// TIA Portal V17 export
// export: Created 2025-03-05T08:02:20.4169739Z, ExportSetting WithDefaults, DisplayName Totally Integrated Automation Portal, DisplayVersion V17 Update 8, DisplayName TIA Portal Openness, DisplayVersion V17 Update 8, DisplayName TIA Portal Version Control Interface, DisplayVersion V17, DisplayName SINAMICS Startdrive Advanced, DisplayVersion V17 SP2, DisplayName SINAMICS Startdrive G110M, G120, G120C, G120D, G120P, G115D, DisplayVersion V17 SP2, DisplayName SINAMICS Startdrive G130, G150, S120, S150, SINAMICS MV, S210, DisplayVersion V17 SP2, DisplayName STEP 7 Professional, DisplayVersion V17 Update 8, DisplayName SINUMERIK ONE STEP 7 Toolbox, DisplayVersion V17 Update 12, DisplayName SINUMERIK 840D sl STEP 7 Toolbox, DisplayVersion V17 Update 12, DisplayName STEP 7 Safety, DisplayVersion V17 Update 6, DisplayName WinCC Advanced, DisplayVersion V17 Update 8
TYPE "OPEN_CLOSE"
// stored: IsFailsafeCompliant false
   STRUCT
      CLOSED_PART_A_I : Bool;   // ADVANCED PART "A" INPUT / CLOSED PART A INPUT
      CLOSED_PART_B_I : Bool;   // ADVANCED PART "B" INPUT / CLOSED PART B INPUT
      CLOSED_PART_C_I : Bool;   // ADVANCED PART "C" INPUT / CLOSED PART C INPUT
      CLOSED_PART_D_I : Bool;   // ADVANCED PART "D" INPUT / CLOSED PART D INPUT
      CLOSED_PRESSURE_SW_1_I : Bool;   // ADVANCED PRESSURE SWITCH 1 / CLOSED PRESSURE SWITCH 1 INPUT
      CLOSED_PRESSURE_SW_2_I : Bool;   // ADVANCED PRESSURE SWITCH 2 / CLOSED PRESSURE SWITCH 2 INPUT
      OPEN_PART_A_I : Bool;   // RETURNED PART "A" INPUT / OPEN PART A INPUT
      OPEN_PART_B_I : Bool;   // RETURNED PART "B" INPUT / OPEN PART B INPUT
      OPEN_PART_C_I : Bool;   // RETURNED PART "C" INPUT / OPEN PART C INPUT
      OPEN_PART_D_I : Bool;   // RETURNED PART "D" INPUT / OPEN PART D INPUT
      OPEN_PRESSURE_SW_1_I : Bool;   // RETURNED PRESSURE SWITCH 1 / OPEN PRESSURE SWITCH 1 INPUT
      OPEN_PRESSURE_SW_2_I : Bool;   // RETURNED PRESSURE SWITCH 2 / OPEN PRESSURE SWITCH 2 INPUT
      CLOSED_LOW_PRESSURE_SW_I : Bool;   // CLOSED LOW PRESSURE SWITCH INPUT
      OPEN_LOW_PRESSURE_SW_I : Bool;   // OPEN LOW PRESSURE SWITCH INPUT
      ANY_CLOSED : Bool;   // ANY CLOSED INPUT
      ANY_OPEN : Bool;   // ANY OPEN INPUT
      GENERAL_CONDITIONS : Bool;   // GENERAL CONDITIONS
      CLOSE_CONDITIONS : Bool;   // ADVANCE CONDITIONS / CLOSE CONDITIONS
      OPEN_CONDITIONS : Bool;   // RETURN CONDITIONS / OPEN CONDITIONS
      RELEASE_PRESSURE_CONDITIONS : Bool;   // RELIEVE PRESSURE CONDITIONS / RELEASE PRESSURE CONDITIONS
      LOW_PRESSURE_CONDITIONS : Bool;   // RELIEVE PRESSURE CONDITIONS / LOW PRESSURE CONDITIONS
      GENERAL_CONDITIONS_HELP : Bool;   // GENERAL CONDITIONS HELP
      CLOSE_CONDITIONS_HELP : Bool;   // CLOSE CONDITIONS HELP
      OPEN_CONDITIONS_HELP : Bool;   // OPEN CONDITIONS HELP
      RELEASE_PRESSURE_CONDITIONS_HELP : Bool;   // RELEASE PRESSURE CONDITIONS HELP
      LOW_PRESSURE_CONDITIONS_HELP : Bool;   // LOW PRESSURE CONDITIONS HELP
      CLOSE_MANUAL_REQUEST : Bool;   // ADVANCE MANUAL REQUEST / CLOSE MANUAL REQUEST
      OPEN_MANUAL_REQUEST : Bool;   // RETURN MANUAL REQUEST / OPEN MANUAL REQUEST
      RELEASE_PRESSURE_MANUAL_REQUEST : Bool;   // RELIEVE PRESSURE MANUAL REQUEST / RELEASE PRESSURE MANUAL REQUEST
      LOW_PRESSURE_MANUAL_REQUEST : Bool;   // RELIEVE PRESSURE MANUAL REQUEST / LOW PRESSURE MANUAL REQUEST
      CLOSE_AUTO_REQUEST : Bool;   // ADVANCE AUTO REQUEST / CLOSE AUTO REQUEST
      OPEN_AUTO_REQUEST : Bool;   // RETURN AUTO REQUEST / OPEN AUTO REQUEST
      RELEASE_PRESSURE_AUTO_REQUEST : Bool;   // RELIEVE PRESSURE AUTO REQUEST / RELEASE PRESSURE AUTO REQUEST
      LOW_PRESSURE_AUTO_REQUEST : Bool;   // LOW PRESSURE AUTO REQUEST
      CLOSE_GLOBAL_REQUEST : Bool;   // ADVANCE GLOBAL REQUEST / CLOSE GLOBAL REQUEST
      OPEN_GLOBAL_REQUEST : Bool;   // RETURN GLOBAL REQUEST / OPEN GLOBAL REQUEST
      RELEASE_PRESSURE_GLOBAL_REQUEST : Bool;   // RELIEVE PRESSURE GLOBAL REQUEST / RELEASE PRESSURE GLOBAL REQUEST
      LOW_PRESSURE_GLOBAL_REQUEST : Bool;   // LOW PRESSURE GLOBAL REQUEST
      CLOSE_COMMAND : Bool;   // ADVANCE COMMAND / CLOSE COMMAND
      OPEN_COMMAND : Bool;   // RETURN COMMAND / OPEN COMMAND
      RELEASE_PRESSURE_COMMAND : Bool;   // RELIEVE PRESSURE COMMAND / RELEASE PRESSURE COMMAND
      CLOSE_LOW_PRESSURE_COMMAND : Bool;   // CLOSE LOW PRESSURE COMMAND
      OPEN_LOW_PRESSURE_COMMAND : Bool;   // OPEN LOW PRESSURE COMMAND
      CLOSE_LOW_PRESSURE : Bool;   // CLOSE LOW PRESSURE
      OPEN_LOW_PRESSURE : Bool;   // OPEN LOW PRESSURE
      FULL_CLOSED : Bool;   // ADVANCE / CLOSED AND COMMANDED
      FULL_OPEN : Bool;   // RETURN / OPEN AND COMMANDED
      FULL_LOW_PRESSURED : Bool;   // LOW PRESSURED AND COMMANDED
      CHECK_CLOSED : Bool;   // CHECK CLOSED AND COMMANDED
      CHECK_OPEN : Bool;   // CHECK OPEN AND COMMANDED
      CHECK_LOW_PRESSURED : Bool;   // CHECK LOW PRESSURED AND COMMANDED
      SIMULTANEITY_ALARM : Bool;   // SIMULTANEITY FAULT / SIMULTANEITY ALARM
      TIME_EXCEEDED_ALARM : Bool;   // TIME EXCEEDED / TIME EXCEEDED ALARM
      ANY_ACTIVE_ALARM : Bool;   // FAULT / ANY ACTIVE ALARM
      RHP_SEOC_ALARMS : Bool;   // RETURN HOME POSITION AND STOP END OF CYCLE ALARMS
      HMI_ACTD_LOW_AUX : Bool;   // HMI FLOWMETER SCREEN CLOSED LOW AUXILIARY
      HMI_DEACTD_LOW_AUX : Bool;   // HMI FLOWMETER SCREEN OPEN LOW AUXILIARY
      PULSE_1 : Bool;   // AUXILIAR ADVANCED PRESSURE SWITCH 1 FAULT / PULSE 1
      PULSE_2 : Bool;   // AUXILIAR ADVANCED PRESSURE SWITCH 2 FAULT / PULSE 2
      PULSE_3 : Bool;   // AUXILIAR RETURNED PRESSURE SWITCH 1 FAULT / PULSE 3
      PULSE_4 : Bool;   // AUXILIAR RETURNED PRESSURE SWITCH 2 FAULT / PULSE 4
      PULSE_5 : Bool;   // AUXILIAR RETURNED PRESSURE SWITCH 1 FAULT / PULSE 5
      PULSE_6 : Bool;   // AUXILIAR RETURNED PRESSURE SWITCH 2 FAULT / PULSE 6
      PULSE_7 : Bool;   // AUXILIAR RETURNED PRESSURE SWITCH 1 FAULT / PULSE 7
      PULSE_8 : Bool;   // AUXILIAR RETURNED PRESSURE SWITCH 2 FAULT / PULSE 8
   END_STRUCT;
END_TYPE
